// LS Electric XG5000 project: interlock
// PLC LSPLC
// module base 0 slot 0: 입출력 모듈:XBC-DR30S (DC 24V 입력 18점, 릴레이 출력 12점)

PROGRAM interlock (task: 스캔 프로그램)

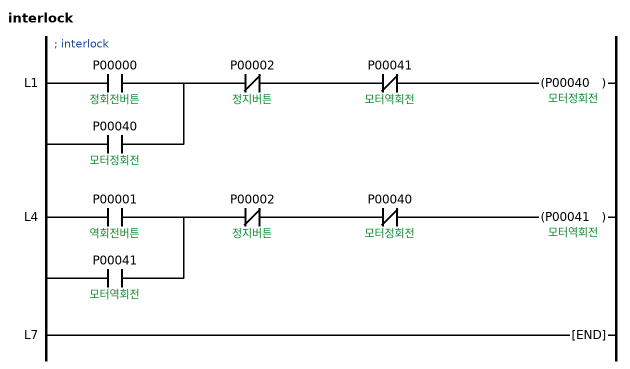
// interlock
; L1
LOAD      P00000	// 정회전버튼
OR        P00040	// 모터정회전
AND NOT   P00002	// 정지버튼
AND NOT   P00041	// 모터역회전
OUT       P00040	// 모터정회전
; L4
LOAD      P00001	// 역회전버튼
OR        P00041	// 모터역회전
AND NOT   P00002	// 정지버튼
AND NOT   P00040	// 모터정회전
OUT       P00041	// 모터역회전
; L7
END